// TIA Portal V17 export
// export: Created 2024-06-25T12:57:18.4905673Z, ExportSetting WithDefaults, DisplayName Totally Integrated Automation Portal, DisplayVersion V17 Update 6, DisplayName TIA Portal Openness, DisplayVersion V17 Update 6, DisplayName TIA Portal Version Control Interface, DisplayVersion V17, DisplayName STEP 7 Professional, DisplayVersion V17 Update 6, DisplayName STEP 7 Safety, DisplayVersion V17 Update 6, DisplayName WinCC Advanced, DisplayVersion V17 Update 6
FUNCTION "Llavin Filtrado" : Void   // FC3, LAD
{ S7_Optimized_Access := 'TRUE' }
VERSION : 0.1
// stored: AutoNumber true, IsIECCheckEnabled false, SetENOAutomatically false, UDAEnableTagReadback false
BEGIN

REGION Network 1: LLAVIN A MAN/LOC
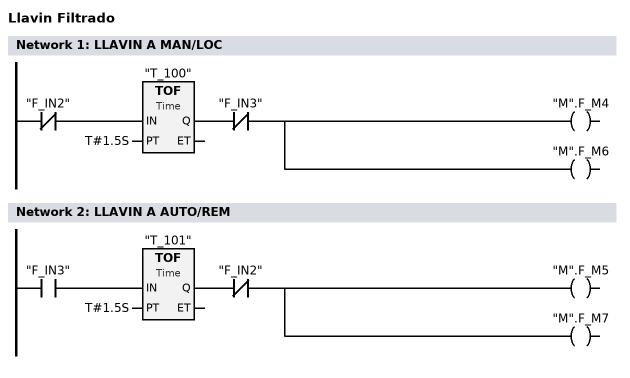
   RUNG wire#powerrail
      I_Contact( "F_IN2" )
      { S7_Templates := "time_type := Time" } "T_100".TOF(pt := T#1.5S, et =>)
      I_Contact( "F_IN3" )
      wire#w1
      Coil( "M".F_M4 )
   END_RUNG
   RUNG wire#w1
      Coil( "M".F_M6 )
   END_RUNG
   // the same network as SCL:
   "T_100".TOF(IN := NOT "F_IN2", PT := T#1.5S);
   "M".F_M4 := "T_100".Q AND NOT "F_IN3";
   "M".F_M6 := "M".F_M4;
END_REGION

REGION Network 2: LLAVIN A AUTO/REM
   RUNG wire#powerrail
      Contact( "F_IN3" )
      { S7_Templates := "time_type := Time" } "T_101".TOF(pt := T#1.5S, et =>)
      I_Contact( "F_IN2" )
      wire#w1
      Coil( "M".F_M5 )
   END_RUNG
   RUNG wire#w1
      Coil( "M".F_M7 )
   END_RUNG
   // the same network as SCL:
   "T_101".TOF(IN := "F_IN3", PT := T#1.5S);
   "M".F_M5 := "T_101".Q AND NOT "F_IN2";
   "M".F_M7 := "M".F_M5;
END_REGION
END_FUNCTION
